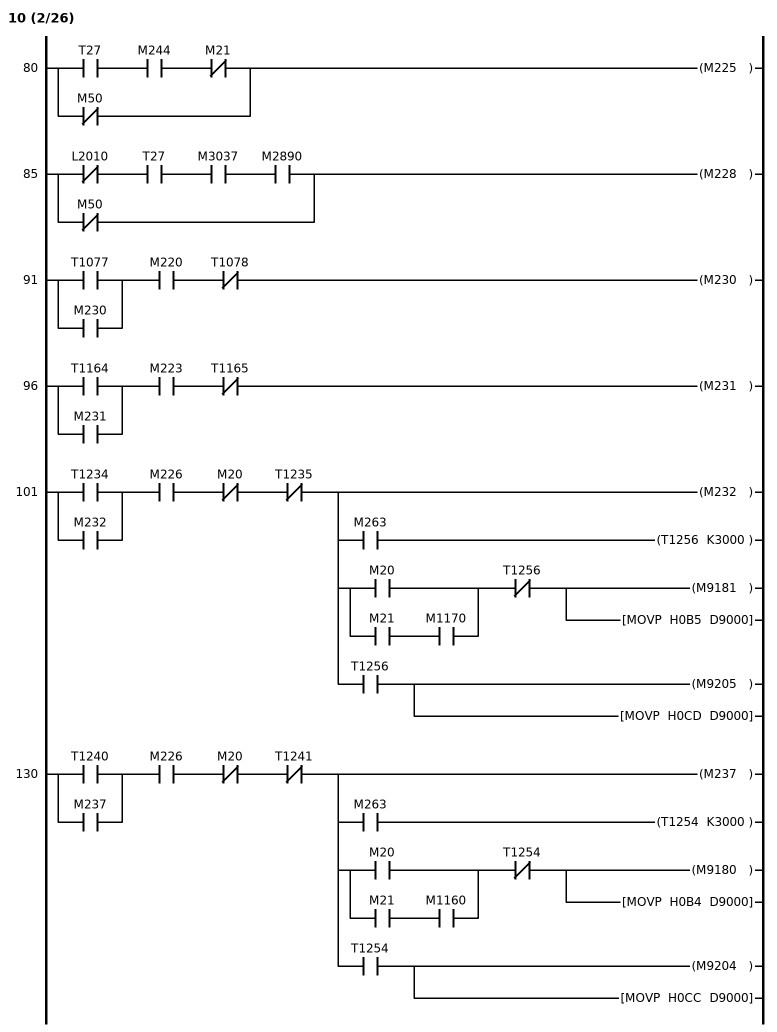
80    LD      T27
      AND     M244
      ANI     M21
      ORI     M50
      OUT     M225
85    LDI     L2010
      AND     T27
      AND     M3037
      AND     M2890
      ORI     M50
      OUT     M228
91    LD      T1077
      OR      M230
      AND     M220
      ANI     T1078
      OUT     M230
96    LD      T1164
      OR      M231
      AND     M223
      ANI     T1165
      OUT     M231
101   LD      T1234
      OR      M232
      AND     M226
      ANI     M20
      ANI     T1235
      OUT     M232
      MPS
      AND     M263
      OUT     T1256 K3000
      MRD
      LD      M20
      LD      M21
      AND     M1170
      ORB
      ANB
      ANI     T1256
      OUT     M9181
      MOVP    H0B5 D9000
      MPP
      AND     T1256
      OUT     M9205
      MOVP    H0CD D9000
130   LD      T1240
      OR      M237
      AND     M226
      ANI     M20
      ANI     T1241
      OUT     M237
      MPS
      AND     M263
      OUT     T1254 K3000
      MRD
      LD      M20
      LD      M21
      AND     M1160
      ORB
      ANB
      ANI     T1254
      OUT     M9180
      MOVP    H0B4 D9000
      MPP
      AND     T1254
      OUT     M9204
      MOVP    H0CC D9000
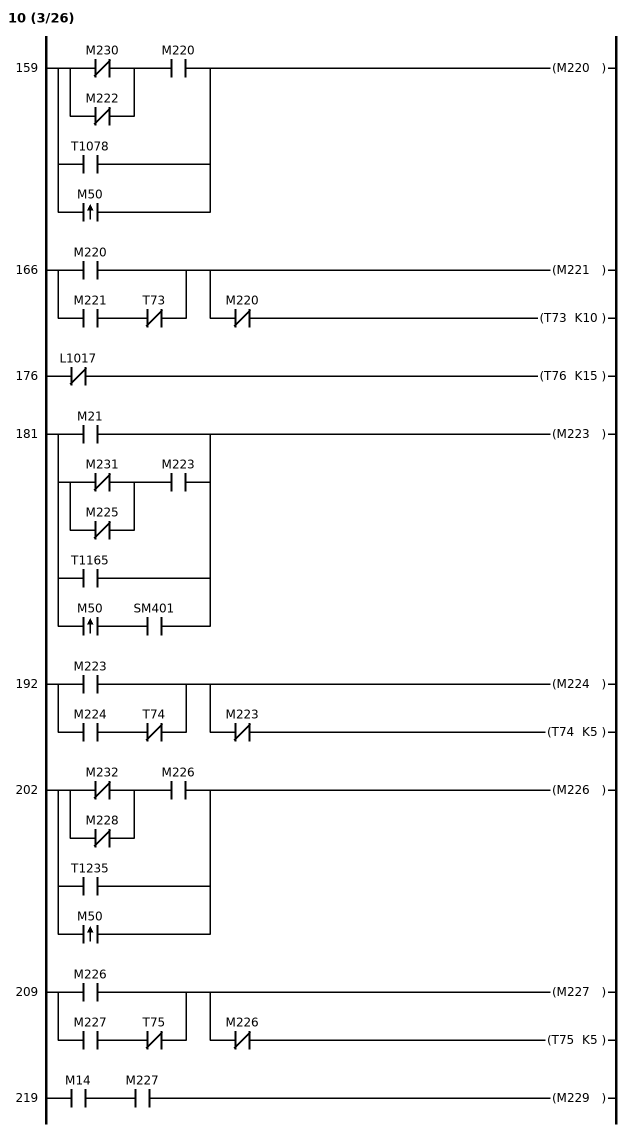
159   LDI     M230
      ORI     M222
      AND     M220
      OR      T1078
      ORP     M50
      OUT     M220
166   LD      M220
      LD      M221
      ANI     T73
      ORB
      OUT     M221
      ANI     M220
      OUT     T73 K10
176   LDI     L1017
      OUT     T76 K15
181   LD      M21
      LDI     M231
      ORI     M225
      AND     M223
      ORB
      OR      T1165
      LDP     M50
      AND     SM401
      ORB
      OUT     M223
192   LD      M223
      LD      M224
      ANI     T74
      ORB
      OUT     M224
      ANI     M223
      OUT     T74 K5
202   LDI     M232
      ORI     M228
      AND     M226
      OR      T1235
      ORP     M50
      OUT     M226
209   LD      M226
      LD      M227
      ANI     T75
      ORB
      OUT     M227
      ANI     M226
      OUT     T75 K5
219   LD      M14
      AND     M227
      OUT     M229
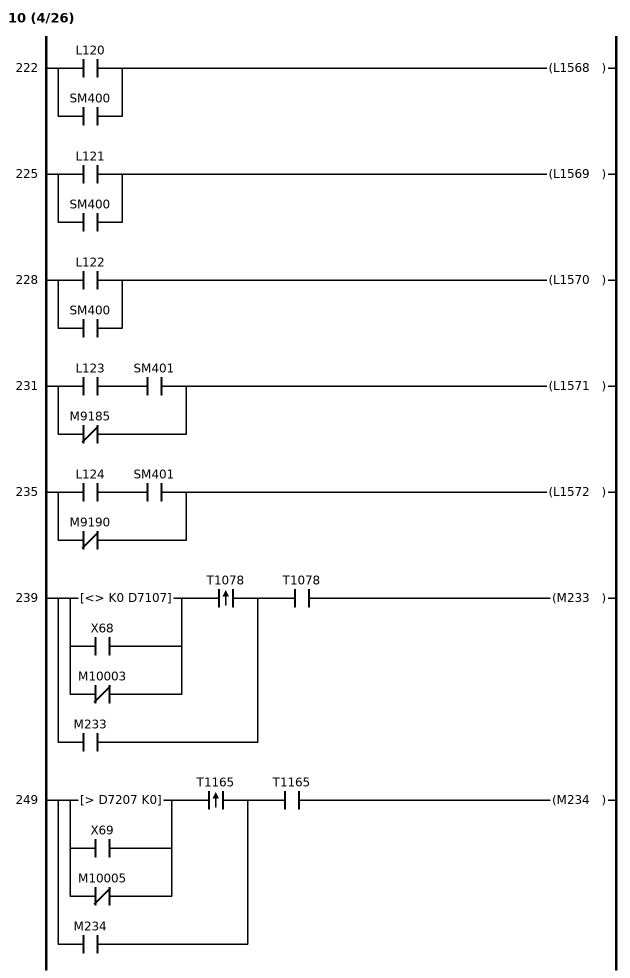
222   LD      L120
      OR      SM400
      OUT     L1568
225   LD      L121
      OR      SM400
      OUT     L1569
228   LD      L122
      OR      SM400
      OUT     L1570
231   LD      L123
      AND     SM401
      ORI     M9185
      OUT     L1571
235   LD      L124
      AND     SM401
      ORI     M9190
      OUT     L1572
239   LD<>    K0 D7107
      OR      X68
      ORI     M10003
      ANDP    T1078
      OR      M233
      AND     T1078
      OUT     M233
249   LD>     D7207 K0
      OR      X69
      ORI     M10005
      ANDP    T1165
      OR      M234
      AND     T1165
      OUT     M234
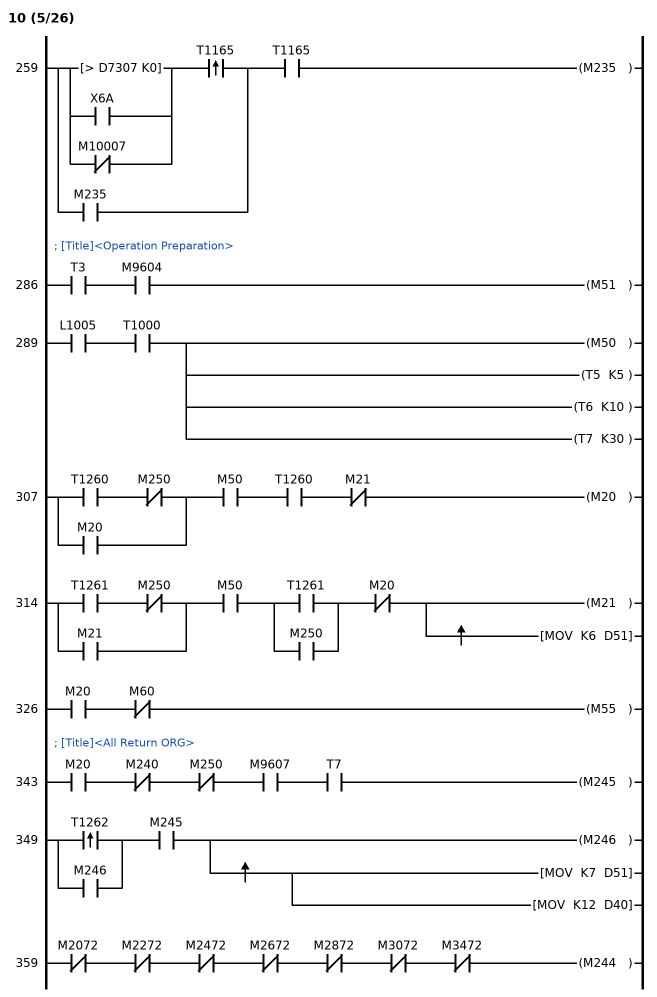
259   LD>     D7307 K0
      OR      X6A
      ORI     M10007
      ANDP    T1165
      OR      M235
      AND     T1165
      OUT     M235
; [Title]<Operation Preparation>
286   LD      T3
      AND     M9604
      OUT     M51
289   LD      L1005
      AND     T1000
      OUT     M50
      OUT     T5 K5
      OUT     T6 K10
      OUT     T7 K30
; 
; 
; 
307   LD      T1260
      ANI     M250
      OR      M20
      AND     M50
      AND     T1260
      ANI     M21
      OUT     M20
314   LD      T1261
      ANI     M250
      OR      M21
      AND     M50
      LD      T1261
      OR      M250
      ANB
      ANI     M20
      OUT     M21
      MEP
      MOV     K6 D51
326   LD      M20
      ANI     M60
      OUT     M55
; [Title]<All Return ORG>
343   LD      M20
      ANI     M240
      ANI     M250
      AND     M9607
      AND     T7
      OUT     M245
349   LDP     T1262
      OR      M246
      AND     M245
      OUT     M246
      MEP
      MOV     K7 D51
      MOV     K12 D40
359   LDI     M2072
      ANI     M2272
      ANI     M2472
      ANI     M2672
      ANI     M2872
      ANI     M3072
      ANI     M3472
      OUT     M244
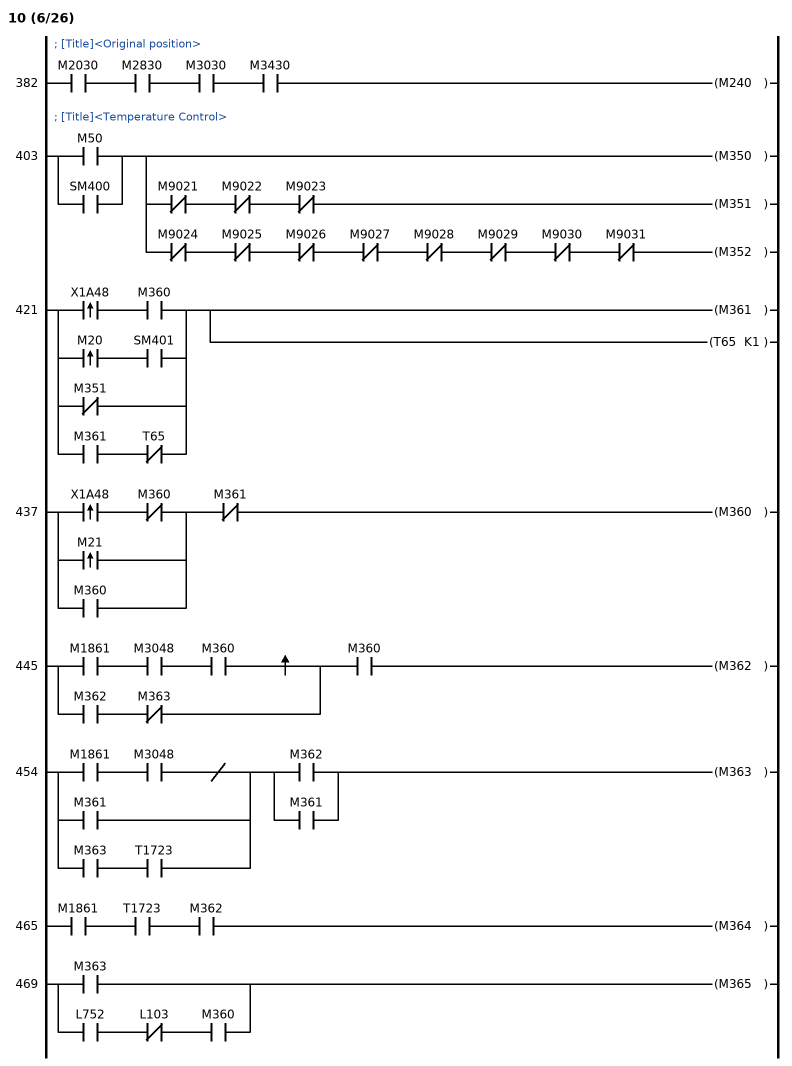
; [Title]<Original position>
382   LD      M2030
      AND     M2830
      AND     M3030
      AND     M3430
      OUT     M240
; [Title]<Temperature Control>
403   LD      M50
      OR      SM400
      OUT     M350
      MPS
      ANI     M9021
      ANI     M9022
      ANI     M9023
      OUT     M351
      MPP
      ANI     M9024
      ANI     M9025
      ANI     M9026
      ANI     M9027
      ANI     M9028
      ANI     M9029
      ANI     M9030
      ANI     M9031
      OUT     M352
421   LDP     X1A48
      AND     M360
      LDP     M20
      AND     SM401
      ORB
      ORI     M351
      LD      M361
      ANI     T65
      ORB
      OUT     M361
      OUT     T65 K1
437   LDP     X1A48
      ANI     M360
      ORP     M21
      OR      M360
      ANI     M361
      OUT     M360
445   LD      M1861
      AND     M3048
      AND     M360
      MEP
      LD      M362
      ANI     M363
      ORB
      AND     M360
      OUT     M362
454   LD      M1861
      AND     M3048
      INV
      OR      M361
      LD      M363
      AND     T1723
      ORB
      LD      M362
      OR      M361
      ANB
      OUT     M363
465   LD      M1861
      AND     T1723
      AND     M362
      OUT     M364
469   LD      M363
      LD      L752
      ANI     L103
      AND     M360
      ORB
      OUT     M365
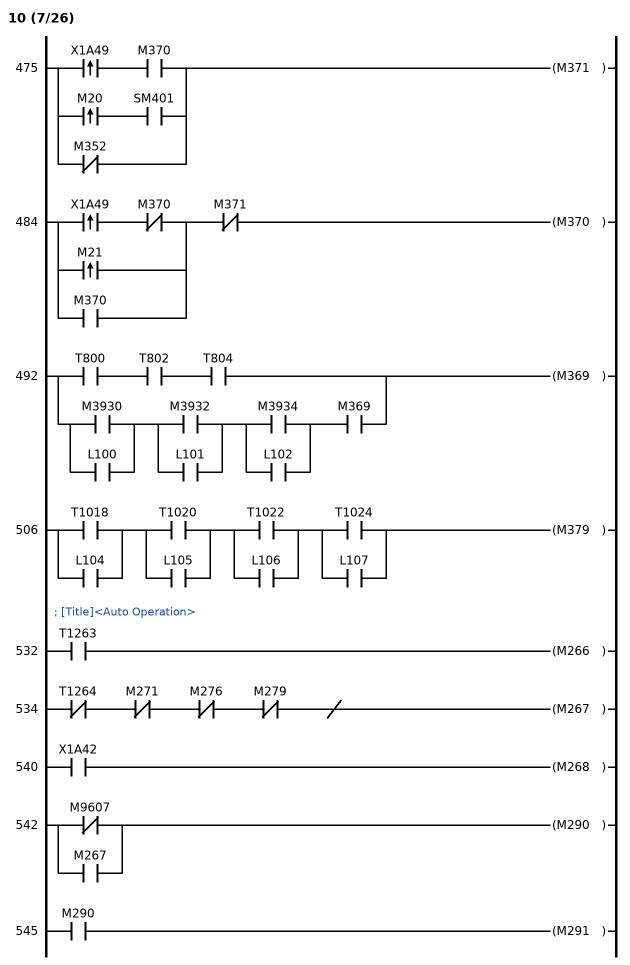
475   LDP     X1A49
      AND     M370
      LDP     M20
      AND     SM401
      ORB
      ORI     M352
      OUT     M371
484   LDP     X1A49
      ANI     M370
      ORP     M21
      OR      M370
      ANI     M371
      OUT     M370
492   LD      T800
      AND     T802
      AND     T804
      LD      M3930
      OR      L100
      LD      M3932
      OR      L101
      ANB
      LD      M3934
      OR      L102
      ANB
      AND     M369
      ORB
      OUT     M369
506   LD      T1018
      OR      L104
      LD      T1020
      OR      L105
      ANB
      LD      T1022
      OR      L106
      ANB
      LD      T1024
      OR      L107
      ANB
      OUT     M379
; [Title]<Auto Operation>
532   LD      T1263
      OUT     M266
534   LDI     T1264
      ANI     M271
      ANI     M276
      ANI     M279
      INV
      OUT     M267
540   LD      X1A42
      OUT     M268
542   LDI     M9607
      OR      M267
      OUT     M290
545   LD      M290
      OUT     M291
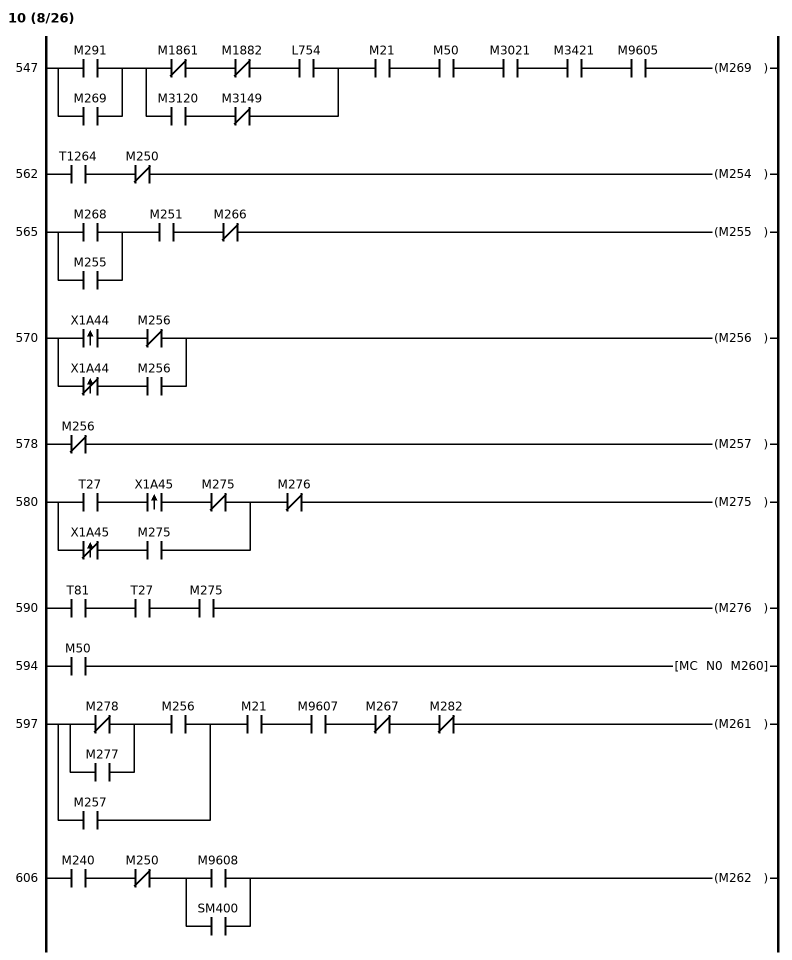
547   LD      M291
      OR      M269
      LDI     M1861
      ANI     M1882
      AND     L754
      LD      M3120
      ANI     M3149
      ORB
      ANB
      AND     M21
      AND     M50
      AND     M3021
      AND     M3421
      AND     M9605
      OUT     M269
562   LD      T1264
      ANI     M250
      OUT     M254
565   LD      M268
      OR      M255
      AND     M251
      ANI     M266
      OUT     M255
570   LDP     X1A44
      ANI     M256
      LDPI    X1A44
      AND     M256
      ORB
      OUT     M256
578   LDI     M256
      OUT     M257
580   LD      T27
      ANDP    X1A45
      ANI     M275
      LDPI    X1A45
      AND     M275
      ORB
      ANI     M276
      OUT     M275
590   LD      T81
      AND     T27
      AND     M275
      OUT     M276
594   LD      M50
      MC      N0 M260
597   LDI     M278
      OR      M277
      AND     M256
      OR      M257
      AND     M21
      AND     M9607
      ANI     M267
      ANI     M282
      OUT     M261
606   LD      M240
      ANI     M250
      LD      M9608
      OR      SM400
      ANB
      OUT     M262
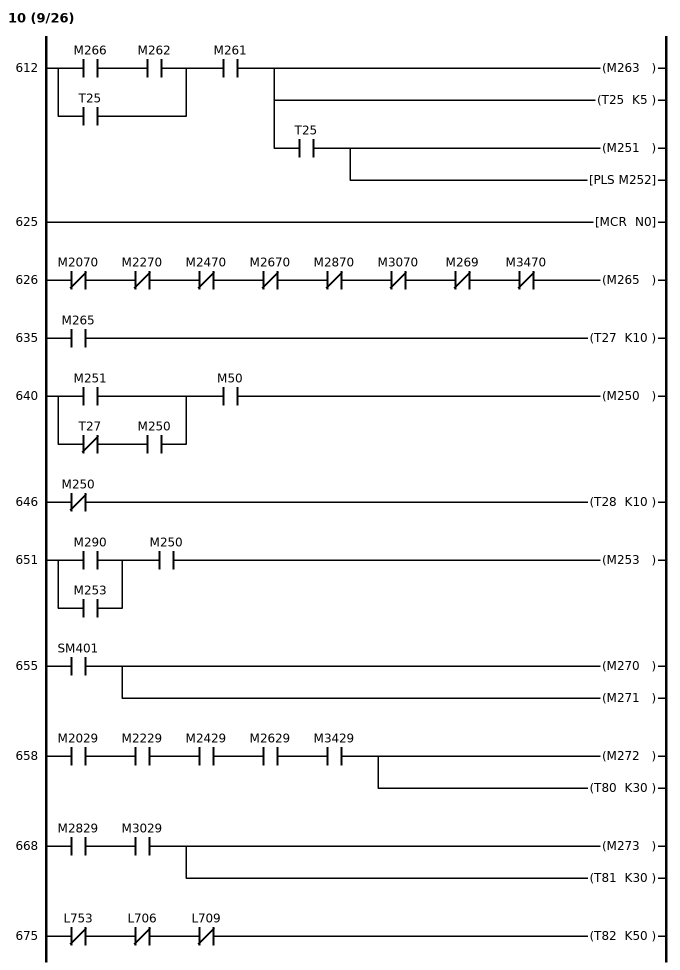
612   LD      M266
      AND     M262
      OR      T25
      AND     M261
      OUT     M263
      OUT     T25 K5
      AND     T25
      OUT     M251
      PLS     M252
625   MCR     N0
626   LDI     M2070
      ANI     M2270
      ANI     M2470
      ANI     M2670
      ANI     M2870
      ANI     M3070
      ANI     M269
      ANI     M3470
      OUT     M265
635   LD      M265
      OUT     T27 K10
640   LD      M251
      LDI     T27
      AND     M250
      ORB
      AND     M50
      OUT     M250
646   LDI     M250
      OUT     T28 K10
651   LD      M290
      OR      M253
      AND     M250
      OUT     M253
655   LD      SM401
      OUT     M270
      OUT     M271
658   LD      M2029
      AND     M2229
      AND     M2429
      AND     M2629
      AND     M3429
      OUT     M272
      OUT     T80 K30
668   LD      M2829
      AND     M3029
      OUT     M273
      OUT     T81 K30
675   LDI     L753
      ANI     L706
      ANI     L709
      OUT     T82 K50
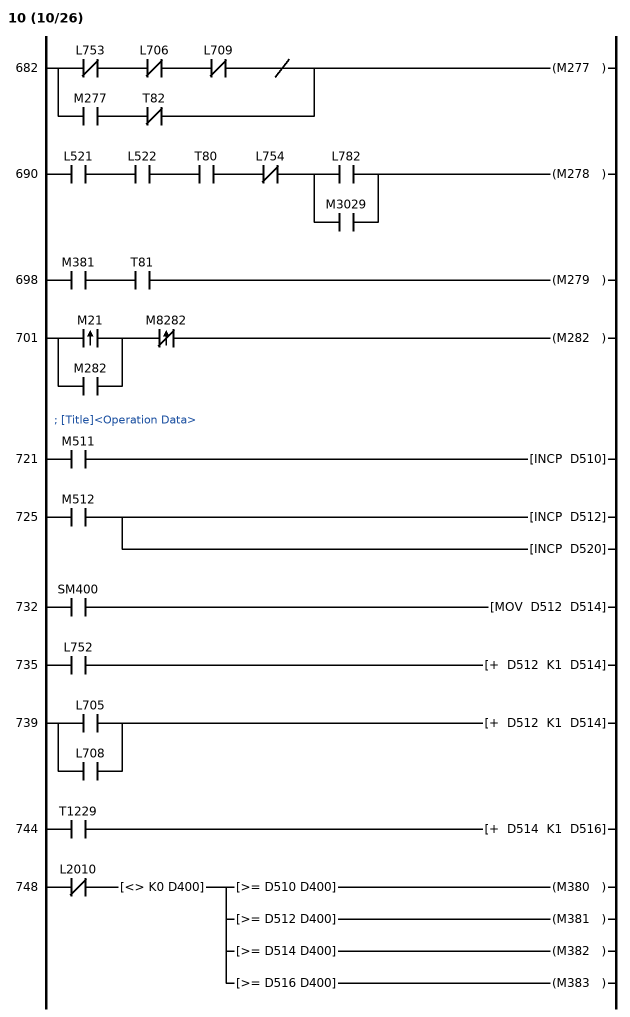
682   LDI     L753
      ANI     L706
      ANI     L709
      INV
      LD      M277
      ANI     T82
      ORB
      OUT     M277
690   LD      L521
      AND     L522
      AND     T80
      ANI     L754
      LD      L782
      OR      M3029
      ANB
      OUT     M278
698   LD      M381
      AND     T81
      OUT     M279
701   LDP     M21
      OR      M282
      ANDPI   M8282
      OUT     M282
; [Title]<Operation Data>
721   LD      M511
      INCP    D510
725   LD      M512
      INCP    D512
      INCP    D520
732   LD      SM400
      MOV     D512 D514
735   LD      L752
      +       D512 K1 D514
739   LD      L705
      OR      L708
      +       D512 K1 D514
744   LD      T1229
      +       D514 K1 D516
748   LDI     L2010
      AND<>   K0 D400
      MPS
      AND>=   D510 D400
      OUT     M380
      MRD
      AND>=   D512 D400
      OUT     M381
      MRD
      AND>=   D514 D400
      OUT     M382
      MPP
      AND>=   D516 D400
      OUT     M383
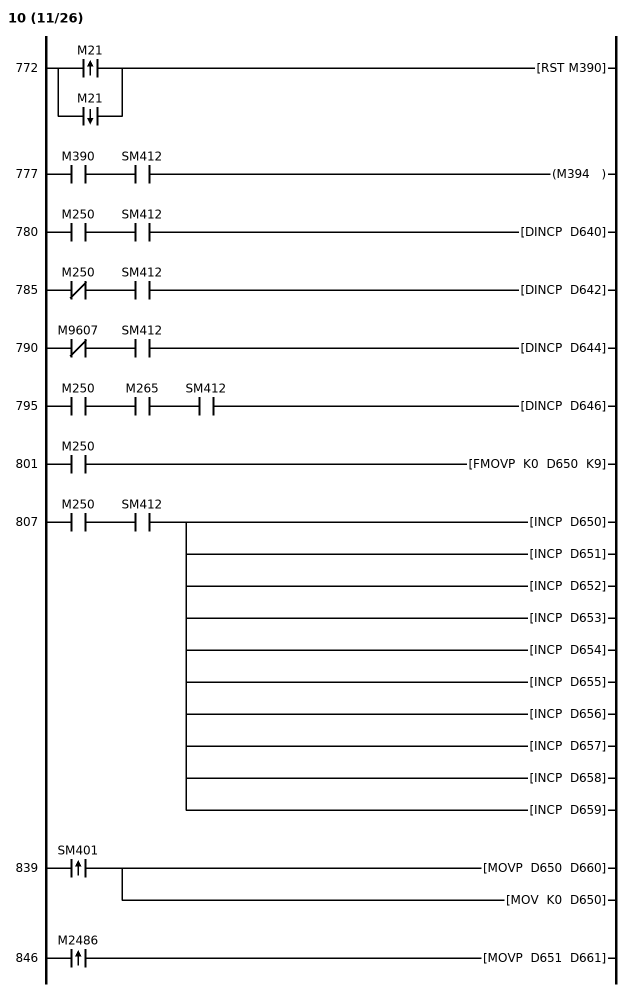
772   LDP     M21
      ORF     M21
      RST     M390
777   LD      M390
      AND     SM412
      OUT     M394
780   LD      M250
      AND     SM412
      DINCP   D640
785   LDI     M250
      AND     SM412
      DINCP   D642
790   LDI     M9607
      AND     SM412
      DINCP   D644
795   LD      M250
      AND     M265
      AND     SM412
      DINCP   D646
801   LD      M250
      FMOVP   K0 D650 K9
807   LD      M250
      AND     SM412
      INCP    D650
      INCP    D651
      INCP    D652
      INCP    D653
      INCP    D654
      INCP    D655
      INCP    D656
      INCP    D657
      INCP    D658
      INCP    D659
839   LDP     SM401
      MOVP    D650 D660
      MOV     K0 D650
846   LDP     M2486
      MOVP    D651 D661
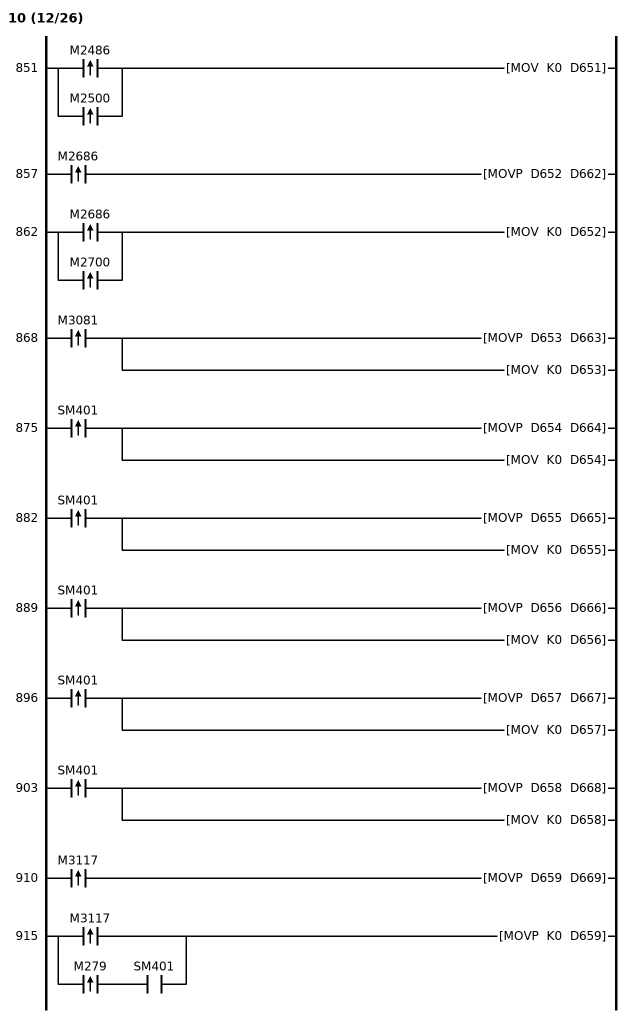
851   LDP     M2486
      ORP     M2500
      MOV     K0 D651
857   LDP     M2686
      MOVP    D652 D662
862   LDP     M2686
      ORP     M2700
      MOV     K0 D652
868   LDP     M3081
      MOVP    D653 D663
      MOV     K0 D653
875   LDP     SM401
      MOVP    D654 D664
      MOV     K0 D654
882   LDP     SM401
      MOVP    D655 D665
      MOV     K0 D655
889   LDP     SM401
      MOVP    D656 D666
      MOV     K0 D656
896   LDP     SM401
      MOVP    D657 D667
      MOV     K0 D657
903   LDP     SM401
      MOVP    D658 D668
      MOV     K0 D658
910   LDP     M3117
      MOVP    D659 D669
915   LDP     M3117
      LDP     M279
      AND     SM401
      ORB
      MOVP    K0 D659
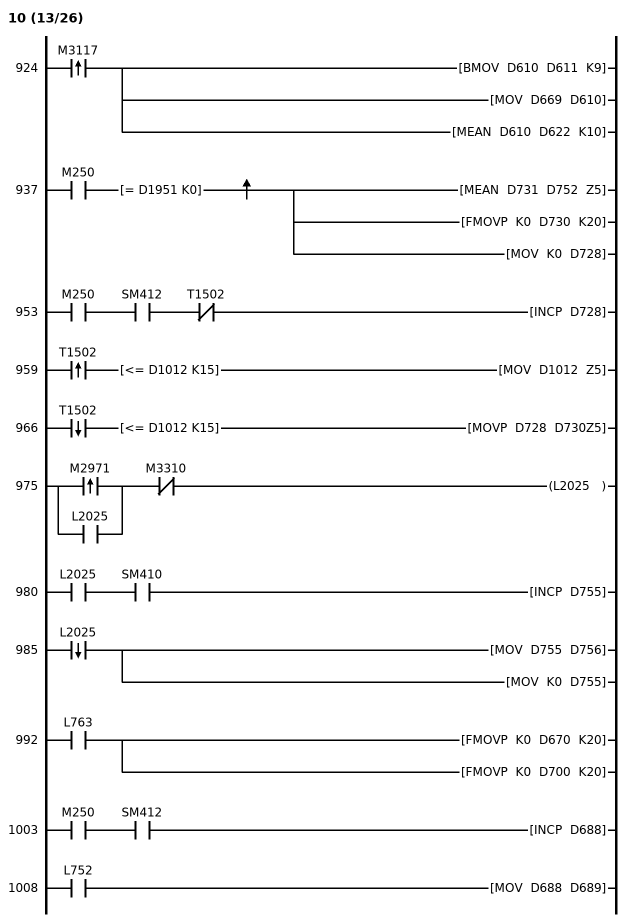
924   LDP     M3117
      BMOV    D610 D611 K9
      MOV     D669 D610
      MEAN    D610 D622 K10
; 
937   LD      M250
      AND=    D1951 K0
      MEP
      MEAN    D731 D752 Z5
      FMOVP   K0 D730 K20
      MOV     K0 D728
953   LD      M250
      AND     SM412
      ANI     T1502
      INCP    D728
959   LDP     T1502
      AND<=   D1012 K15
      MOV     D1012 Z5
966   LDF     T1502
      AND<=   D1012 K15
      MOVP    D728 D730Z5
975   LDP     M2971
      OR      L2025
      ANI     M3310
      OUT     L2025
980   LD      L2025
      AND     SM410
      INCP    D755
985   LDF     L2025
      MOV     D755 D756
      MOV     K0 D755
; 
992   LD      L763
      FMOVP   K0 D670 K20
      FMOVP   K0 D700 K20
1003  LD      M250
      AND     SM412
      INCP    D688
1008  LD      L752
      MOV     D688 D689
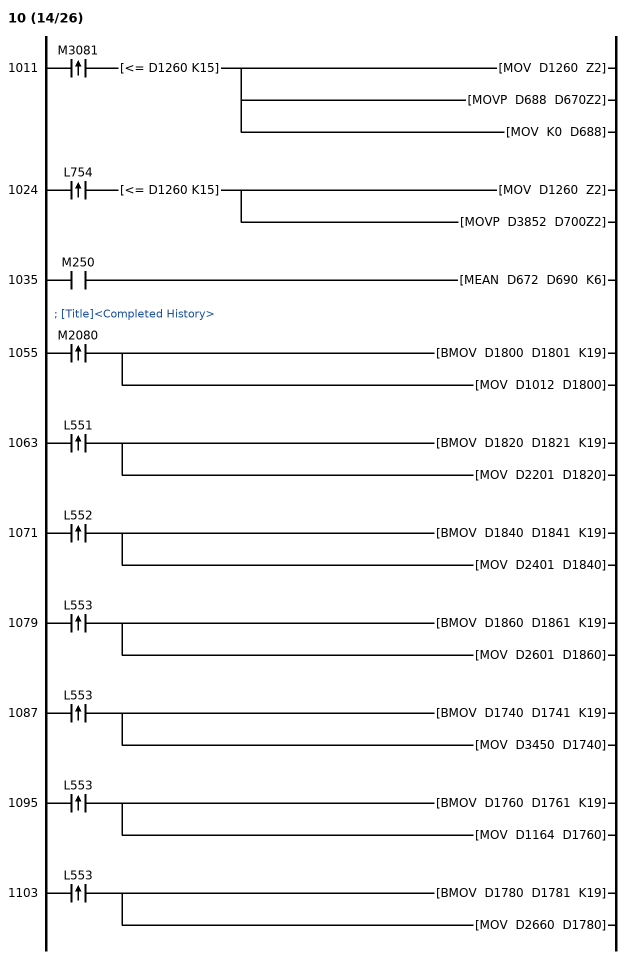
1011  LDP     M3081
      AND<=   D1260 K15
      MOV     D1260 Z2
      MOVP    D688 D670Z2
      MOV     K0 D688
1024  LDP     L754
      AND<=   D1260 K15
      MOV     D1260 Z2
      MOVP    D3852 D700Z2
1035  LD      M250
      MEAN    D672 D690 K6
; [Title]<Completed History>
1055  LDP     M2080
      BMOV    D1800 D1801 K19
      MOV     D1012 D1800
1063  LDP     L551
      BMOV    D1820 D1821 K19
      MOV     D2201 D1820
1071  LDP     L552
      BMOV    D1840 D1841 K19
      MOV     D2401 D1840
1079  LDP     L553
      BMOV    D1860 D1861 K19
      MOV     D2601 D1860
1087  LDP     L553
      BMOV    D1740 D1741 K19
      MOV     D3450 D1740
1095  LDP     L553
      BMOV    D1760 D1761 K19
      MOV     D1164 D1760
1103  LDP     L553
      BMOV    D1780 D1781 K19
      MOV     D2660 D1780
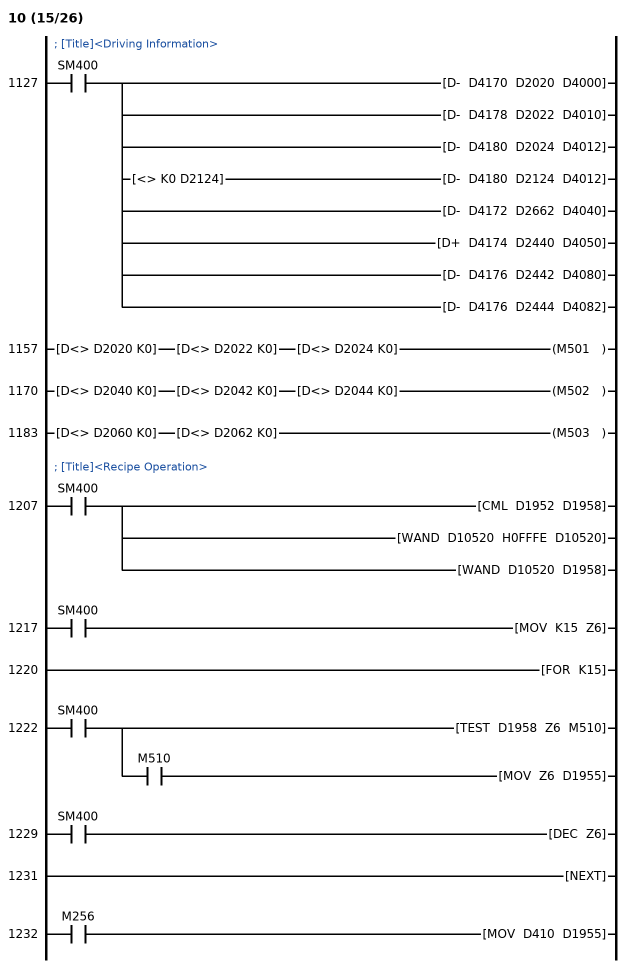
; [Title]<Driving Information>
1127  LD      SM400
      D-      D4170 D2020 D4000
      D-      D4178 D2022 D4010
      D-      D4180 D2024 D4012
      MPS
      AND<>   K0 D2124
      D-      D4180 D2124 D4012
      MPP
      D-      D4172 D2662 D4040
      D+      D4174 D2440 D4050
      D-      D4176 D2442 D4080
      D-      D4176 D2444 D4082
1157  LDD<>   D2020 K0
      ANDD<>  D2022 K0
      ANDD<>  D2024 K0
      OUT     M501
1170  LDD<>   D2040 K0
      ANDD<>  D2042 K0
      ANDD<>  D2044 K0
      OUT     M502
1183  LDD<>   D2060 K0
      ANDD<>  D2062 K0
      OUT     M503
; [Title]<Recipe Operation>
1207  LD      SM400
      CML     D1952 D1958
      WAND    D10520 H0FFFE D10520
      WAND    D10520 D1958
1217  LD      SM400
      MOV     K15 Z6
1220  FOR     K15
1222  LD      SM400
      TEST    D1958 Z6 M510
      AND     M510
      MOV     Z6 D1955
1229  LD      SM400
      DEC     Z6
1231  NEXT
1232  LD      M256
      MOV     D410 D1955
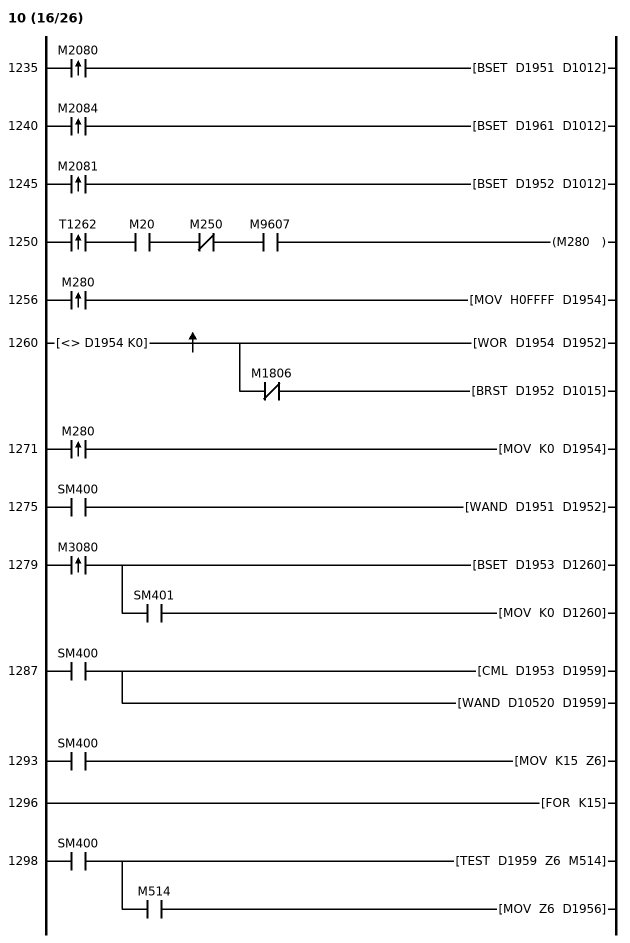
1235  LDP     M2080
      BSET    D1951 D1012
1240  LDP     M2084
      BSET    D1961 D1012
1245  LDP     M2081
      BSET    D1952 D1012
1250  LDP     T1262
      AND     M20
      ANI     M250
      AND     M9607
      OUT     M280
1256  LDP     M280
      MOV     H0FFFF D1954
1260  LD<>    D1954 K0
      MEP
      WOR     D1954 D1952
      ANI     M1806
      BRST    D1952 D1015
1271  LDP     M280
      MOV     K0 D1954
1275  LD      SM400
      WAND    D1951 D1952
1279  LDP     M3080
      BSET    D1953 D1260
      AND     SM401
      MOV     K0 D1260
1287  LD      SM400
      CML     D1953 D1959
      WAND    D10520 D1959
1293  LD      SM400
      MOV     K15 Z6
1296  FOR     K15
1298  LD      SM400
      TEST    D1959 Z6 M514
      AND     M514
      MOV     Z6 D1956
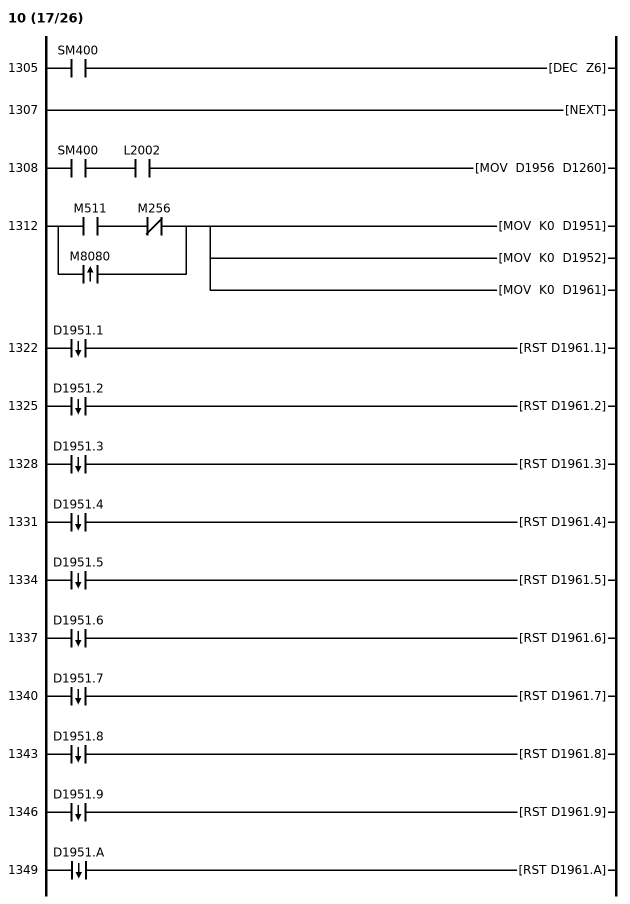
1305  LD      SM400
      DEC     Z6
1307  NEXT
1308  LD      SM400
      AND     L2002
      MOV     D1956 D1260
1312  LD      M511
      ANI     M256
      ORP     M8080
      MOV     K0 D1951
      MOV     K0 D1952
      MOV     K0 D1961
1322  LDF     D1951.1
      RST     D1961.1
1325  LDF     D1951.2
      RST     D1961.2
1328  LDF     D1951.3
      RST     D1961.3
1331  LDF     D1951.4
      RST     D1961.4
1334  LDF     D1951.5
      RST     D1961.5
1337  LDF     D1951.6
      RST     D1961.6
1340  LDF     D1951.7
      RST     D1961.7
1343  LDF     D1951.8
      RST     D1961.8
1346  LDF     D1951.9
      RST     D1961.9
1349  LDF     D1951.A
      RST     D1961.A
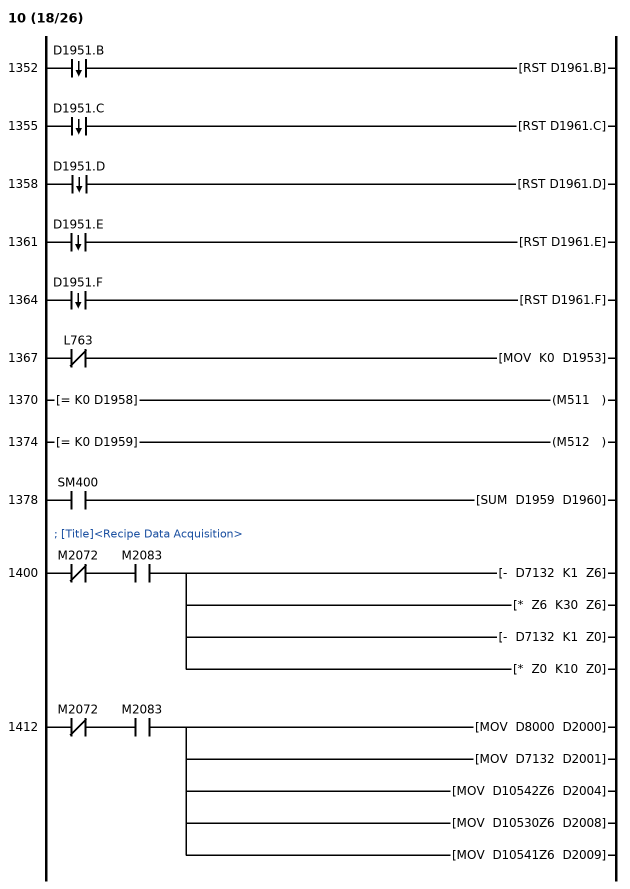
1352  LDF     D1951.B
      RST     D1961.B
1355  LDF     D1951.C
      RST     D1961.C
1358  LDF     D1951.D
      RST     D1961.D
1361  LDF     D1951.E
      RST     D1961.E
1364  LDF     D1951.F
      RST     D1961.F
1367  LDI     L763
      MOV     K0 D1953
1370  LD=     K0 D1958
      OUT     M511
1374  LD=     K0 D1959
      OUT     M512
1378  LD      SM400
      SUM     D1959 D1960
; [Title]<Recipe Data Acquisition>
1400  LDI     M2072
      AND     M2083
      -       D7132 K1 Z6
      *       Z6 K30 Z6
      -       D7132 K1 Z0
      *       Z0 K10 Z0
1412  LDI     M2072
      AND     M2083
      MOV     D8000 D2000
      MOV     D7132 D2001
      MOV     D10542Z6 D2004
      MOV     D10530Z6 D2008
      MOV     D10541Z6 D2009
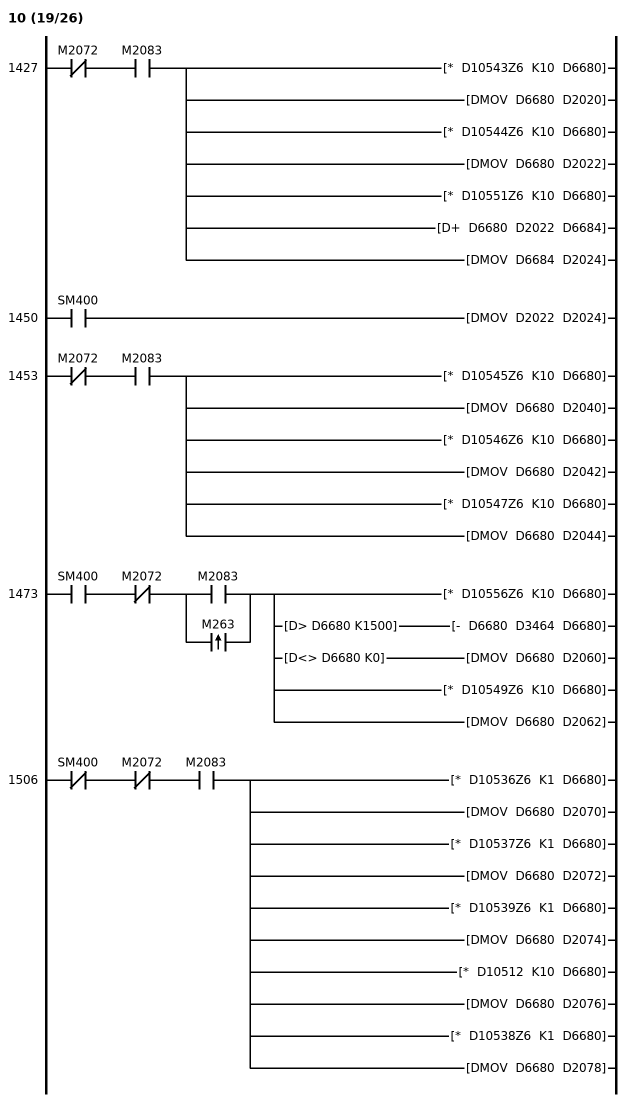
1427  LDI     M2072
      AND     M2083
      *       D10543Z6 K10 D6680
      DMOV    D6680 D2020
      *       D10544Z6 K10 D6680
      DMOV    D6680 D2022
      *       D10551Z6 K10 D6680
      D+      D6680 D2022 D6684
      DMOV    D6684 D2024
1450  LD      SM400
      DMOV    D2022 D2024
1453  LDI     M2072
      AND     M2083
      *       D10545Z6 K10 D6680
      DMOV    D6680 D2040
      *       D10546Z6 K10 D6680
      DMOV    D6680 D2042
      *       D10547Z6 K10 D6680
      DMOV    D6680 D2044
1473  LD      SM400
      ANI     M2072
      LD      M2083
      ORP     M263
      ANB
      *       D10556Z6 K10 D6680
      MPS
      ANDD>   D6680 K1500
      -       D6680 D3464 D6680
      MRD
      ANDD<>  D6680 K0
      DMOV    D6680 D2060
      MPP
      *       D10549Z6 K10 D6680
      DMOV    D6680 D2062
1506  LDI     SM400
      ANI     M2072
      AND     M2083
      *       D10536Z6 K1 D6680
      DMOV    D6680 D2070
      *       D10537Z6 K1 D6680
      DMOV    D6680 D2072
      *       D10539Z6 K1 D6680
      DMOV    D6680 D2074
      *       D10512 K10 D6680
      DMOV    D6680 D2076
      *       D10538Z6 K1 D6680
      DMOV    D6680 D2078
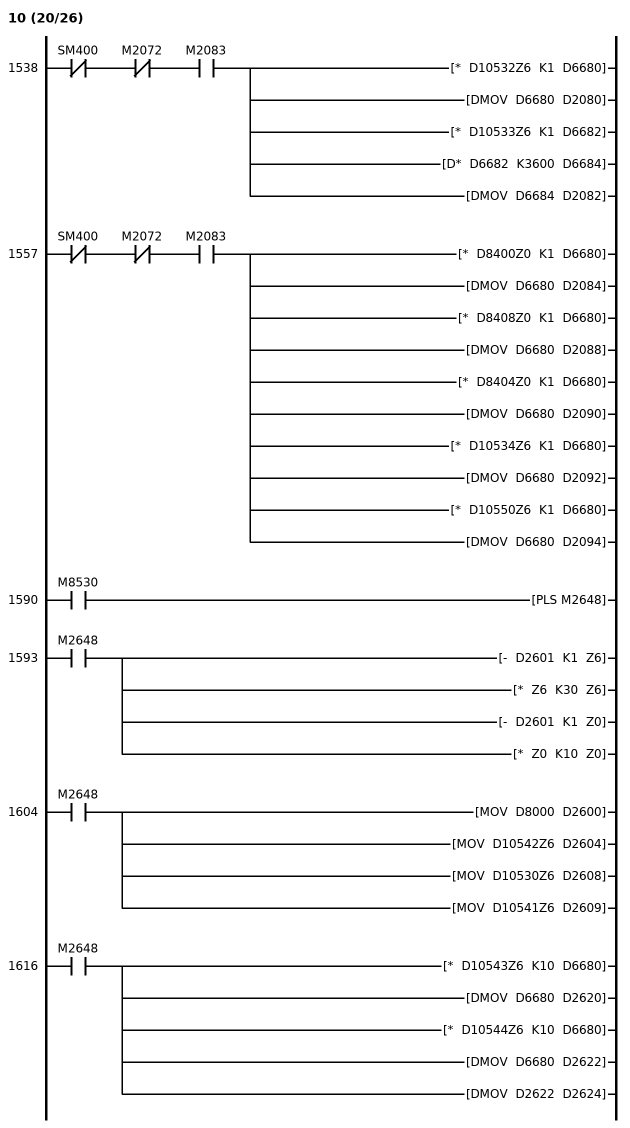
1538  LDI     SM400
      ANI     M2072
      AND     M2083
      *       D10532Z6 K1 D6680
      DMOV    D6680 D2080
      *       D10533Z6 K1 D6682
      D*      D6682 K3600 D6684
      DMOV    D6684 D2082
1557  LDI     SM400
      ANI     M2072
      AND     M2083
      *       D8400Z0 K1 D6680
      DMOV    D6680 D2084
      *       D8408Z0 K1 D6680
      DMOV    D6680 D2088
      *       D8404Z0 K1 D6680
      DMOV    D6680 D2090
      *       D10534Z6 K1 D6680
      DMOV    D6680 D2092
      *       D10550Z6 K1 D6680
      DMOV    D6680 D2094
1590  LD      M8530
      PLS     M2648
1593  LD      M2648
      -       D2601 K1 Z6
      *       Z6 K30 Z6
      -       D2601 K1 Z0
      *       Z0 K10 Z0
1604  LD      M2648
      MOV     D8000 D2600
      MOV     D10542Z6 D2604
      MOV     D10530Z6 D2608
      MOV     D10541Z6 D2609
1616  LD      M2648
      *       D10543Z6 K10 D6680
      DMOV    D6680 D2620
      *       D10544Z6 K10 D6680
      DMOV    D6680 D2622
      DMOV    D2622 D2624
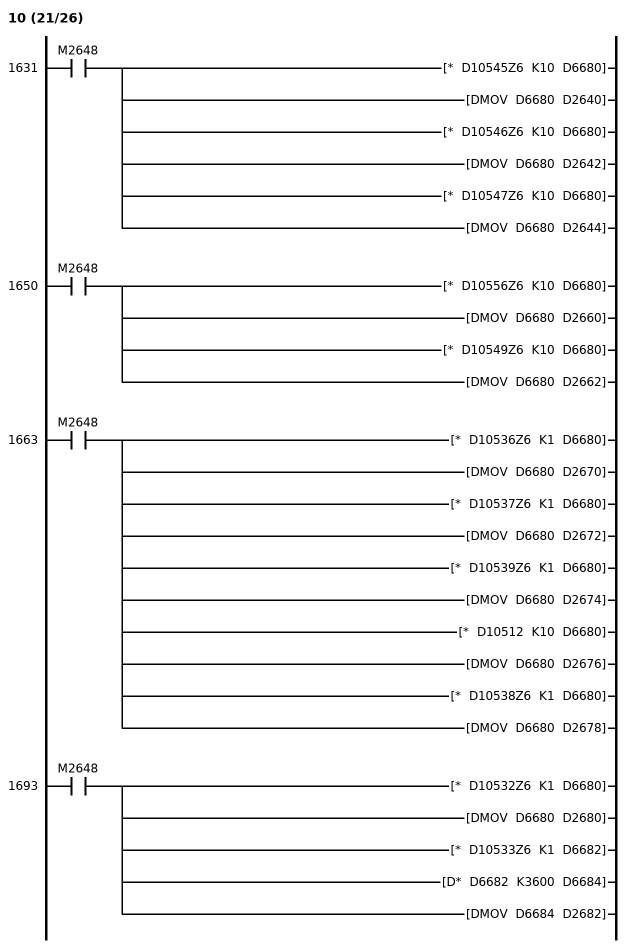
1631  LD      M2648
      *       D10545Z6 K10 D6680
      DMOV    D6680 D2640
      *       D10546Z6 K10 D6680
      DMOV    D6680 D2642
      *       D10547Z6 K10 D6680
      DMOV    D6680 D2644
1650  LD      M2648
      *       D10556Z6 K10 D6680
      DMOV    D6680 D2660
      *       D10549Z6 K10 D6680
      DMOV    D6680 D2662
1663  LD      M2648
      *       D10536Z6 K1 D6680
      DMOV    D6680 D2670
      *       D10537Z6 K1 D6680
      DMOV    D6680 D2672
      *       D10539Z6 K1 D6680
      DMOV    D6680 D2674
      *       D10512 K10 D6680
      DMOV    D6680 D2676
      *       D10538Z6 K1 D6680
      DMOV    D6680 D2678
1693  LD      M2648
      *       D10532Z6 K1 D6680
      DMOV    D6680 D2680
      *       D10533Z6 K1 D6682
      D*      D6682 K3600 D6684
      DMOV    D6684 D2682
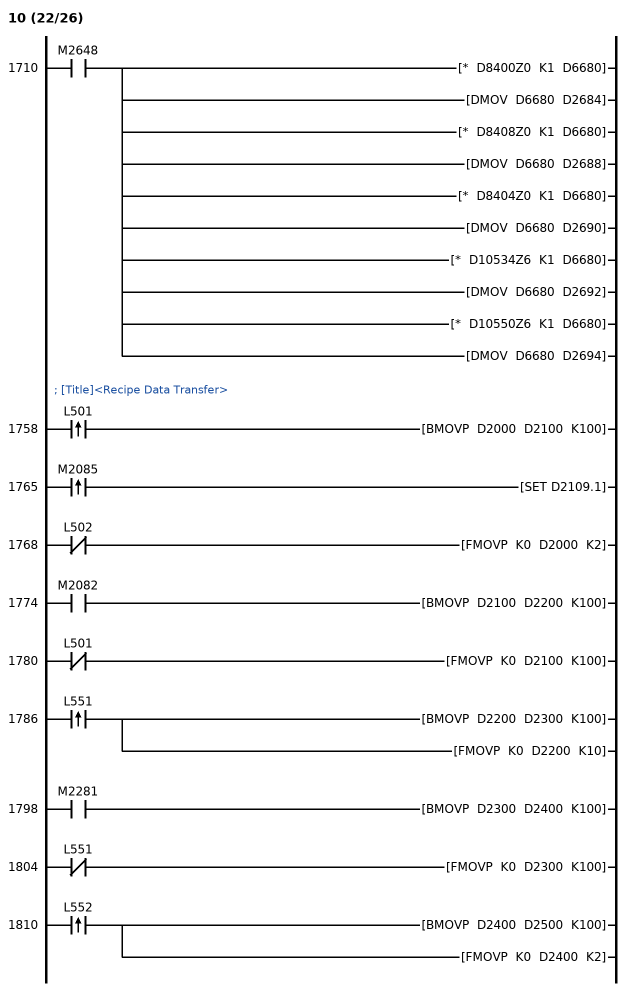
1710  LD      M2648
      *       D8400Z0 K1 D6680
      DMOV    D6680 D2684
      *       D8408Z0 K1 D6680
      DMOV    D6680 D2688
      *       D8404Z0 K1 D6680
      DMOV    D6680 D2690
      *       D10534Z6 K1 D6680
      DMOV    D6680 D2692
      *       D10550Z6 K1 D6680
      DMOV    D6680 D2694
; [Title]<Recipe Data Transfer>
1758  LDP     L501
      BMOVP   D2000 D2100 K100
1765  LDP     M2085
      SET     D2109.1
1768  LDI     L502
      FMOVP   K0 D2000 K2
1774  LD      M2082
      BMOVP   D2100 D2200 K100
1780  LDI     L501
      FMOVP   K0 D2100 K100
1786  LDP     L551
      BMOVP   D2200 D2300 K100
      FMOVP   K0 D2200 K10
1798  LD      M2281
      BMOVP   D2300 D2400 K100
1804  LDI     L551
      FMOVP   K0 D2300 K100
1810  LDP     L552
      BMOVP   D2400 D2500 K100
      FMOVP   K0 D2400 K2
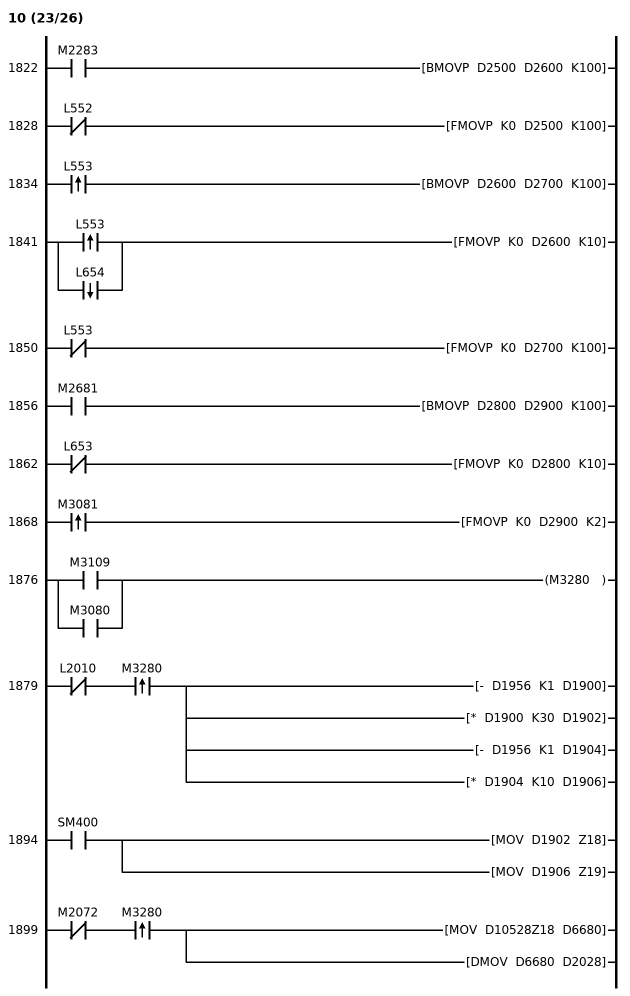
1822  LD      M2283
      BMOVP   D2500 D2600 K100
1828  LDI     L552
      FMOVP   K0 D2500 K100
1834  LDP     L553
      BMOVP   D2600 D2700 K100
1841  LDP     L553
      ORF     L654
      FMOVP   K0 D2600 K10
1850  LDI     L553
      FMOVP   K0 D2700 K100
1856  LD      M2681
      BMOVP   D2800 D2900 K100
1862  LDI     L653
      FMOVP   K0 D2800 K10
1868  LDP     M3081
      FMOVP   K0 D2900 K2
; 
1876  LD      M3109
      OR      M3080
      OUT     M3280
1879  LDI     L2010
      ANDP    M3280
      -       D1956 K1 D1900
      *       D1900 K30 D1902
      -       D1956 K1 D1904
      *       D1904 K10 D1906
1894  LD      SM400
      MOV     D1902 Z18
      MOV     D1906 Z19
1899  LDI     M2072
      ANDP    M3280
      MOV     D10528Z18 D6680
      DMOV    D6680 D2028
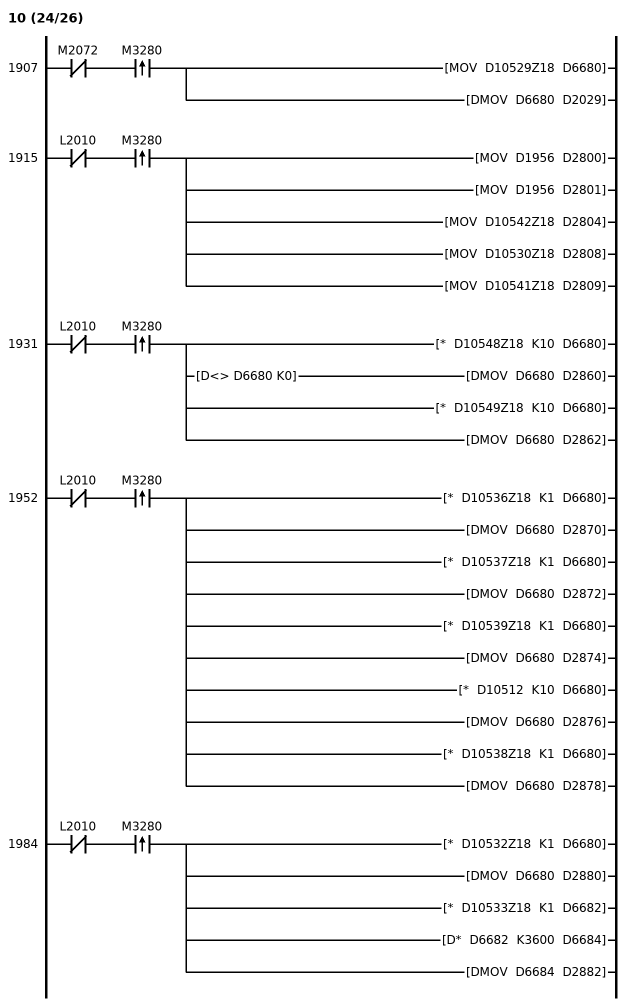
1907  LDI     M2072
      ANDP    M3280
      MOV     D10529Z18 D6680
      DMOV    D6680 D2029
1915  LDI     L2010
      ANDP    M3280
      MOV     D1956 D2800
      MOV     D1956 D2801
      MOV     D10542Z18 D2804
      MOV     D10530Z18 D2808
      MOV     D10541Z18 D2809
1931  LDI     L2010
      ANDP    M3280
      *       D10548Z18 K10 D6680
      MPS
      ANDD<>  D6680 K0
      DMOV    D6680 D2860
      MPP
      *       D10549Z18 K10 D6680
      DMOV    D6680 D2862
1952  LDI     L2010
      ANDP    M3280
      *       D10536Z18 K1 D6680
      DMOV    D6680 D2870
      *       D10537Z18 K1 D6680
      DMOV    D6680 D2872
      *       D10539Z18 K1 D6680
      DMOV    D6680 D2874
      *       D10512 K10 D6680
      DMOV    D6680 D2876
      *       D10538Z18 K1 D6680
      DMOV    D6680 D2878
1984  LDI     L2010
      ANDP    M3280
      *       D10532Z18 K1 D6680
      DMOV    D6680 D2880
      *       D10533Z18 K1 D6682
      D*      D6682 K3600 D6684
      DMOV    D6684 D2882
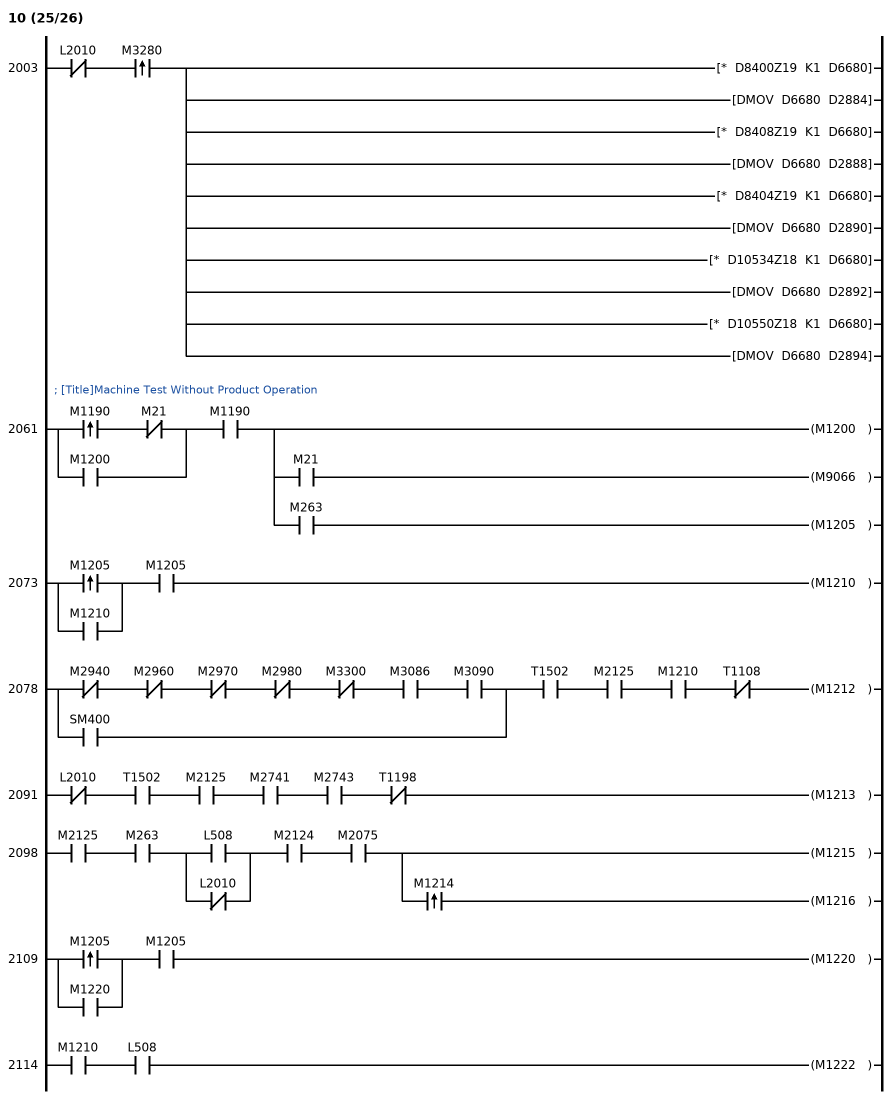
2003  LDI     L2010
      ANDP    M3280
      *       D8400Z19 K1 D6680
      DMOV    D6680 D2884
      *       D8408Z19 K1 D6680
      DMOV    D6680 D2888
      *       D8404Z19 K1 D6680
      DMOV    D6680 D2890
      *       D10534Z18 K1 D6680
      DMOV    D6680 D2892
      *       D10550Z18 K1 D6680
      DMOV    D6680 D2894
; [Title]Machine Test Without Product Operation
2061  LDP     M1190
      ANI     M21
      OR      M1200
      AND     M1190
      OUT     M1200
      MPS
      AND     M21
      OUT     M9066
      MPP
      AND     M263
      OUT     M1205
2073  LDP     M1205
      OR      M1210
      AND     M1205
      OUT     M1210
2078  LDI     M2940
      ANI     M2960
      ANI     M2970
      ANI     M2980
      ANI     M3300
      AND     M3086
      AND     M3090
      OR      SM400
      AND     T1502
      AND     M2125
      AND     M1210
      ANI     T1108
      OUT     M1212
2091  LDI     L2010
      AND     T1502
      AND     M2125
      AND     M2741
      AND     M2743
      ANI     T1198
      OUT     M1213
2098  LD      M2125
      AND     M263
      LD      L508
      ORI     L2010
      ANB
      AND     M2124
      AND     M2075
      OUT     M1215
      ANDP    M1214
      OUT     M1216
2109  LDP     M1205
      OR      M1220
      AND     M1205
      OUT     M1220
2114  LD      M1210
      AND     L508
      OUT     M1222
